PROGRAM MAIN
VAR
	Start: BOOL;
	Reset: BOOL;
	Stop: BOOL;
	
	StartLight: BOOL;
	ResetLight: BOOL;
	StopLight: BOOL;
	
	AtBufferEntry : BOOL;
	AtBufferExit : BOOL;
	AtExit : BOOL;
	
	Emitter : BOOL;
	EntryConveyor: BOOL;
	ExitConveyor: BOOL;
	EmergencyStop: BOOL;
	
	isStopON: BOOL;
	isEmgStopON: BOOL;
	isSystemON: BOOL;
	isResetON: BOOL;
	wasEmgBtnPressed: BOOL;
	
	ButtonController : ButtonController;
	EmitterController : EmitterController;
	ConveyorController : ConveyorController;
END_VAR

// I/O Assignments
GVL.mb_Input_Coils[1] := StartLight;
GVL.mb_Input_Coils[2] := ResetLight;
GVL.mb_Input_Coils[3] := StopLight;
GVL.mb_Input_Coils[4] := EntryConveyor;
GVL.mb_Input_Coils[5] := ExitConveyor;
GVL.mb_Input_Coils[6] := Emitter;

AtBufferEntry := GVL.mb_Output_Coils[0];
AtBufferExit := GVL.mb_Output_Coils[1];
AtExit := GVL.mb_Output_Coils[2];
Start := gvl.mb_Output_Coils[3];
Reset := gvl.mb_Output_Coils[4];
Stop := gvl.mb_Output_Coils[5];
EmergencyStop := gvl.mb_Output_Coils[7];
// -------------
//Button Control
ButtonController(StartButton := Start, ResetButton := Reset, StopButton := Stop, 
EmgStopButton := EmergencyStop, StartLight => StartLight, ResetLight => ResetLight, StopLight => StopLight);
// -------------
// Emitter Control
EmitterController(AtBufferEntry := AtBufferEntry, Emitter => Emitter);
// -------------
// Conveyor control
ConveyorController(AtBufferEntry := AtBufferEntry, AtBufferExit := AtBufferExit, AtExit := AtExit, EntryConveyor => EntryConveyor, ExitConveyor => ExitConveyor);
// -------------

END_PROGRAM

(* stored: Version 1.1.0.1, ProductVersion 3.1.4024.12
   POU MAIN: Id {6e8692c7-591f-4c2f-bfee-a5270370c477}, SpecialFunc None *)
